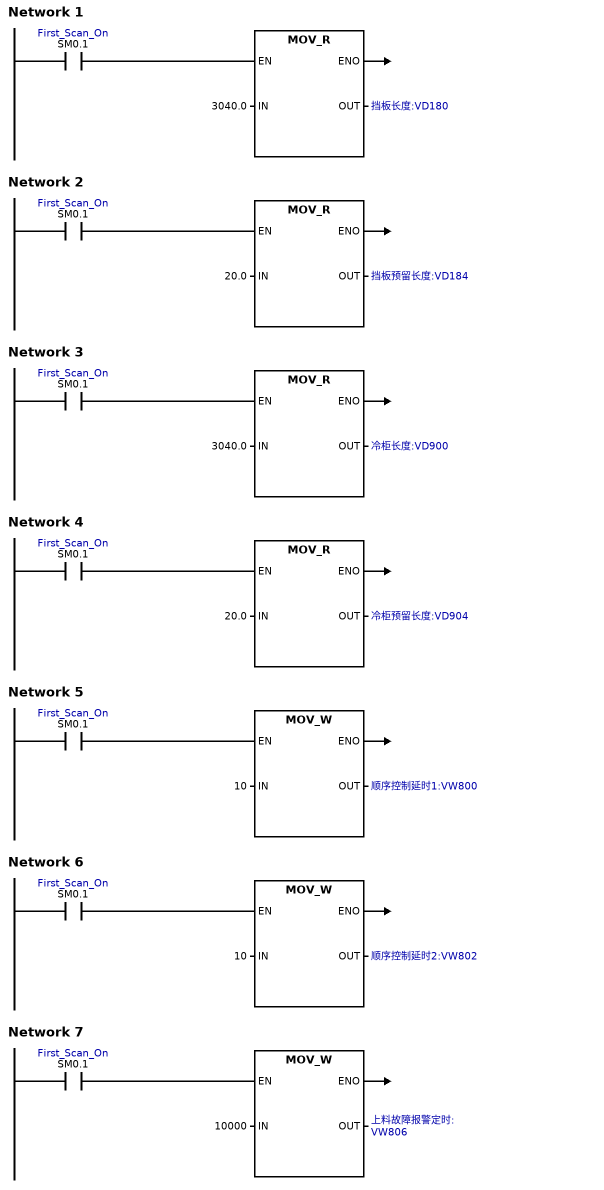
[picture p24: SBR20 networks 1-7]
Network 1
LD     First_Scan_On:SM0.1
MOVR   3040.0, 挡板长度:VD180
Network 2
LD     First_Scan_On:SM0.1
MOVR   20.0, 挡板预留长度:VD184
Network 3
LD     First_Scan_On:SM0.1
MOVR   3040.0, 冷柜长度:VD900
Network 4
LD     First_Scan_On:SM0.1
MOVR   20.0, 冷柜预留长度:VD904
Network 5
LD     First_Scan_On:SM0.1
MOVW   10, 顺序控制延时1:VW800
Network 6
LD     First_Scan_On:SM0.1
MOVW   10, 顺序控制延时2:VW802
Network 7
LD     First_Scan_On:SM0.1
MOVW   10000, 上料故障报警定时:VW806
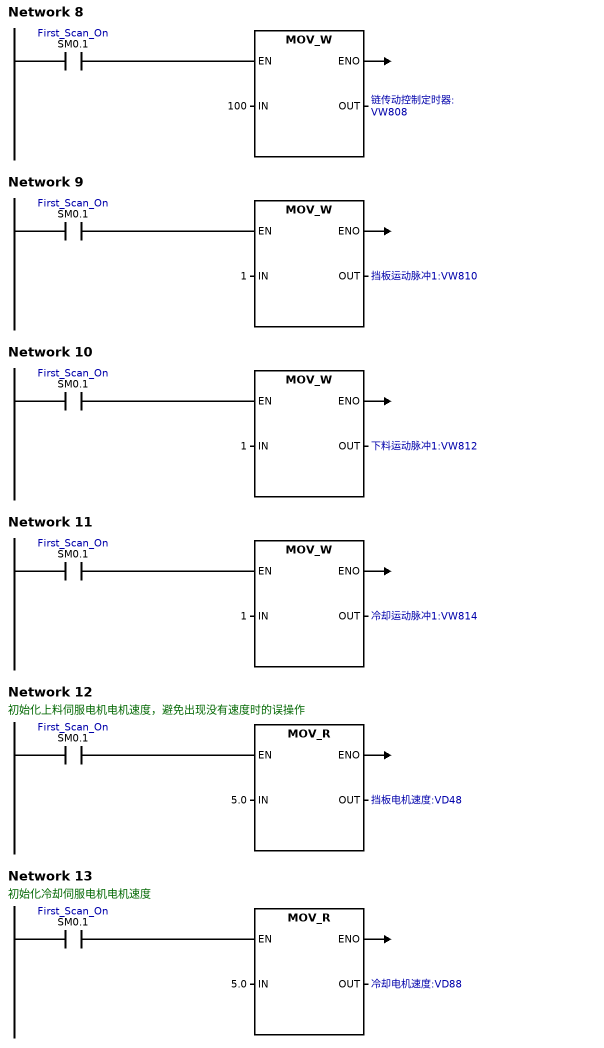
Network 8
LD     First_Scan_On:SM0.1
MOVW   100, 链传动控制定时器:VW808
Network 9
LD     First_Scan_On:SM0.1
MOVW   1, 挡板运动脉冲1:VW810
Network 10
LD     First_Scan_On:SM0.1
MOVW   1, 下料运动脉冲1:VW812
Network 11
LD     First_Scan_On:SM0.1
MOVW   1, 冷却运动脉冲1:VW814
Network 12
// 初始化上料伺服电机电机速度，避免出现没有速度时的误操作
LD     First_Scan_On:SM0.1
MOVR   5.0, 挡板电机速度:VD48
Network 13
// 初始化冷却伺服电机电机速度
LD     First_Scan_On:SM0.1
MOVR   5.0, 冷却电机速度:VD88
END_SUBROUTINE_BLOCK

SUBROUTINE_BLOCK 故障报警:SBR21
TITLE=子程序注释
BEGIN
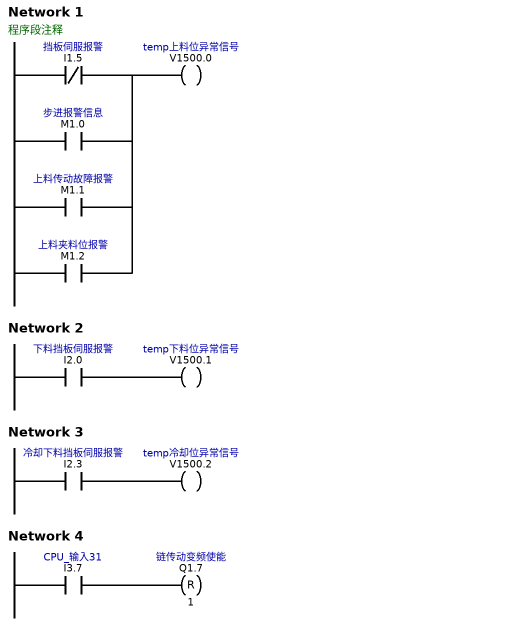
Network 1
// 程序段注释
LDN    挡板伺服报警:I1.5
O      步进报警信息:M1.0
O      上料传动故障报警:M1.1
O      上料夹料位报警:M1.2
=      temp上料位异常信号:V1500.0
Network 2
LD     下料挡板伺服报警:I2.0
=      temp下料位异常信号:V1500.1
Network 3
LD     冷却下料挡板伺服报警:I2.3
=      temp冷却位异常信号:V1500.2
Network 4
LD     CPU_输入31:I3.7
R      链传动变频使能:Q1.7, 1
END_SUBROUTINE_BLOCK
